ABB RAPID module: TCTM831_CYCLE_PATH_FOLLOW_CYCLE.mod

MODULE TCTM831_CYCLE_PATH_FOLLOW_CYCLE
    !*****************************************************
    !Project    : P21-100538 COJAFEX
    !Version:     1.0
    !Description:
    !Date:        04-2022
    !Author:      RLZ
    !*****************************************************
    !
    PERS pos OFFSET:=[0,0,0];
    PERS pos OFFSET_REF:=[0,0,0];
    PERS pos offsetprev:=[0,0,0];

    CONST num CALC_COUNTER:=71;             ! afstand tcp inductie ring - tcp lasers  55
    CONST num POS_FILTER_SIZE:=41;          ! oneven getal was 21
    CONST num ORIENT_FILTER_SIZE:=35;       ! oneven getal was 31
    CONST num PreStartLength:=90;           ! minimaal 2 * POS_FILTER_SIZE
    CONST num MaxLaserOutRange := 10;       ! als laser
    CONST num LaserDistMean := 15;          ! 15 laser datapunten worden gemiddeld voor het bepalen van einde buis (verkleining)
    CONST num EndTubeMinDistance := 12;     ! 20mm gemiddelde afstand verschil tussen de punten voor en de punten na is einde buis

    !PERS num nMovementCounter:=725;         ! Actual tcp heating ring position
    PERS num nPosFilterCounter:=704;        ! Calculated filtered pos position
    PERS num nOrientFilterCounter:=687;     ! Calculated filtered orient position
    PERS pos OrientVectorStart:=[-16.0742,645.886,223.213];
    PERS pos OrientVectorEind:=[-15.8133,665.273,253.56];
    PERS num Lasers{4}:=[-3449.93,-3441.27,-3504.93,-3514.26];
    PERS num nLaserData{4}:=[378.5,383,386.8,377];
    PERS num nLaserDataprev{4}:=[378.5,383,386.8,377];
    PERS num nLaserOutRange{4}:=[0,0,0,0];
    PERS bool END_TUBE_REACHED{2} := [FALSE, FALSE];

    PERS robtarget Assist1;
    PERS robtarget Assist2;
    PERS robtarget Assist3;
    PERS jointtarget joints;
    PERS num As1;
    PERS num As2;
    PERS num As3;
    PERS num As4;
    PERS num As5;
    PERS num As6;
    PERS num As7;

    PERS orient SaveLaserValue{10000};      ! Size should be the same as TargetNew
    PERS orient LaserDataAll{1200}:=[[0,0,0,0],
                                    [0,0,0,0],
                                    [0,0,0,0],
                                    [0,0,0,0],
                                    [0,0,0,0],
                                    [0,0,0,0],
                                    [0,0,0,0],
                                    [0,0,0,0],
                                    [0,0,0,0],
                                    [0,0,0,0],
                                    [0,0,0,0],
                                    [0,0,0,0],
                                    [0,0,0,0],
                                    [0,0,0,0],
                                    [0,0,0,0],
                                    [0,0,0,0],
                                    [0,0,0,0],
                                    [383.5,380.8,383.8,382.3],
                                    [383.5,380.9,383.9,382.2],
                                    [383.6,380.9,383.9,382.2],
                                    [383.6,381,383.8,382.1],
                                    [382.1,380.6,383.9,379.9],
                                    [382.1,380.6,383.9,379.9],
                                    [382.1,380.6,383.9,379.9],
                                    [382.1,380.6,383.8,379.9],
                                    [382.1,380.6,383.8,379.9],
                                    [382.1,380.5,383.7,380],
                                    [382.3,380.5,383.6,380.2],
                                    [382.3,380.3,383.8,380.2],
                                    [382.4,380.3,383.7,380.3],
                                    [382.4,380.4,383.5,380.2],
                                    [382.6,380.5,383.3,380.3],
                                    [382.6,380.6,383.5,380],
                                    [382.7,380.7,383.6,380.1],
                                    [382.8,380.6,383.5,380.1],
                                    [382.8,380.5,383.4,380],
                                    [382.9,380.6,383.3,380.1],
                                    [382.9,380.5,383.3,380.2],
                                    [383,380.4,383.3,380.3],
                                    [383,380.3,383.3,380.3],
                                    [383.1,380.5,383.1,380.3],
                                    [383.1,380.4,383.1,380.3],
                                    [383.2,380.2,383.1,380.4],
                                    [383.2,380.3,382.9,380.4],
                                    [383.2,380.2,383,380.3],
                                    [383.3,380.3,382.9,380.4],
                                    [383.4,380.3,383.1,380.2],
                                    [383.6,380.3,383.1,380.3],
                                    [383.4,380.2,383,380.3],
                                    [383.1,380.3,383.5,380.3],
                                    [383.2,380.3,383.4,380.3],
                                    [383.6,380.4,382.9,380.3],
                                    [383.9,380.3,382.5,380.4],
                                    [383.9,380.3,382.4,380.4],
                                    [383.9,380.4,382.5,380.4],
                                    [384,380.4,382.6,380.5],
                                    [384,380.3,382.6,380.5],
                                    [383,380.9,382.8,379.7],
                                    [383.1,381,382.5,379.4],
                                    [383.1,381.1,382.7,379.5],
                                    [383,381.2,382.7,379.4],
                                    [383,380.9,382.6,379.5],
                                    [382.6,380.7,382.8,379.7],
                                    [382.8,380.6,382.8,379.8],
                                    [382.9,380.3,382.5,380.2],
                                    [383,380.4,382.5,380.1],
                                    [383,380.5,382.8,380],
                                    [383.1,380.6,382.3,379.9],
                                    [383.1,380.6,382.3,379.9],
                                    [383.1,380.7,382.4,379.8],
                                    [383.2,380.6,382.6,379.9],
                                    [383.3,380.5,382.5,379.9],
                                    [383.3,380.5,382.4,380.1],
                                    [383.2,380.4,382.4,380.1],
                                    [383.4,380.3,382.3,380.2],
                                    [383.4,380.2,382.5,380.3],
                                    [383.3,380,382.4,380.3],
                                    [383.3,380.1,382.4,380.4],
                                    [383.6,380,382.6,380.3],
                                    [383.6,380,382.3,380.3],
                                    [383.4,380,382.4,380.4],
                                    [383.4,380.1,382.3,380.5],
                                    [383.3,380,382.3,380.2],
                                    [383.3,380.2,382.3,380.3],
                                    [383.3,380.2,382.5,380.2],
                                    [383.3,380.2,382.6,380.3],
                                    [383.2,380.1,382.4,380.3],
                                    [383.1,380.2,382.5,380.2],
                                    [383,380.1,382.7,380.2],
                                    [383,380.2,382.4,380.1],
                                    [383.1,380.4,383,380],
                                    [382.8,380.3,383.1,380.1],
                                    [382.5,380.4,383.1,379.9],
                                    [382.5,380.5,383.6,379.6],
                                    [382.4,380.7,383.4,379.6],
                                    [382.3,380.9,383.8,379.3],
                                    [382.2,381,383.5,379.2],
                                    [382,381,383.7,379.2],
                                    [381.8,381.1,383.8,379.1],
                                    [381.6,381.3,384.2,378.9],
                                    [381.3,381.3,384.4,378.9],
                                    [381.2,381.4,384.6,378.8],
                                    [381.1,381.4,384.5,378.6],
                                    [380.9,381.6,384.6,378.5],
                                    [380.8,381.6,384.8,378.4],
                                    [380.6,381.7,385.1,378.5],
                                    [380.2,381.9,385.4,378.3],
                                    [380,382.2,385.6,378.2],
                                    [379.7,382.1,385.8,378.2],
                                    [379.4,382.1,386.1,378.2],
                                    [379.5,381.7,386.3,378.2],
                                    [379.5,381.9,386.1,378.4],
                                    [379.5,381.7,386.1,378.4],
                                    [379.5,381.5,386.2,378.6],
                                    [379.3,381.5,386.2,378.6],
                                    [379.3,381.5,386.4,378.6],
                                    [379.3,381.4,386.4,378.6],
                                    [379.2,381.2,386.6,378.7],
                                    [379.1,381.5,386.4,378.9],
                                    [379.1,381.3,386.6,378.8],
                                    [379.1,381.2,386.6,378.9],
                                    [379,381.5,386.5,378.9],
                                    [379,381.4,386.4,378.7],
                                    [378.9,381.3,386.4,378.8],
                                    [378.9,381.2,386.2,379.1],
                                    [378.8,381.1,386.5,378.9],
                                    [378.7,381.1,386.6,378.9],
                                    [378.6,381.2,386.7,379],
                                    [378.5,381.4,386.7,378.8],
                                    [378.5,381.3,386.7,378.8],
                                    [378.4,381.3,387.4,378.8],
                                    [378.4,381.4,387.3,378.6],
                                    [378.3,381.5,387.1,378.6],
                                    [378.3,381.4,387.1,378.5],
                                    [378.2,381.5,387.2,378.5],
                                    [378.4,381.7,387.1,378.4],
                                    [378.4,381.7,387.2,378.4],
                                    [378.3,381.9,387.2,378.3],
                                    [378.2,381.8,387.3,378.2],
                                    [378.3,381.8,387.3,378.1],
                                    [378.1,381.9,387.1,378.2],
                                    [378.3,381.8,387.2,378.2],
                                    [378.2,382,387.3,378.2],
                                    [378.2,382.1,387.3,378.1],
                                    [378.2,382,387.1,378.1],
                                    [378.2,382.1,387,377.9],
                                    [378.2,382.1,387.1,378],
                                    [378.2,382.1,387.4,378],
                                    [378.2,382,387,378.1],
                                    [378.2,382.1,387.6,378],
                                    [378.2,382.1,387.2,378.1],
                                    [378.3,382.2,387.1,378],
                                    [378.3,382.1,387.1,377.9],
                                    [378.3,382.3,387.4,378],
                                    [378.3,382.1,387.1,378],
                                    [378.4,382,387.1,378],
                                    [378.4,381.9,386.9,378.1],
                                    [378.4,382.1,387,378],
                                    [378.4,382,387.2,378.2],
                                    [378.3,382.2,387.1,378.2],
                                    [378.4,382.2,387,378.1],
                                    [378.5,382.1,386.9,378.1],
                                    [378.5,382,387.1,378.2],
                                    [378.5,382,387,378.2],
                                    [378.5,382,386.9,378.1],
                                    [378.6,382,386.7,378.1],
                                    [378.6,382,386.8,378],
                                    [378.6,382,386.9,378.1],
                                    [378.6,382,387.1,378.1],
                                    [378.5,382.1,387.1,378],
                                    [378.5,382.2,386.9,377.9],
                                    [378.5,382.2,386.9,377.9],
                                    [378.6,382.2,387.1,377.9],
                                    [378.6,382.3,387.1,377.8],
                                    [378.6,382.5,387,377.9],
                                    [378.6,382.2,386.7,377.9],
                                    [378.5,382.1,386.8,377.8],
                                    [378.5,382.2,386.9,377.9],
                                    [378.5,382.3,387,377.9],
                                    [378.5,382.3,387.3,377.8],
                                    [378.5,382.2,387.2,377.8],
                                    [378.4,382.3,387.2,377.8],
                                    [378.4,382.3,387.3,377.7],
                                    [378.3,382.3,387.4,377.7],
                                    [378.2,382.4,387.4,377.7],
                                    [378.2,382.3,387.5,377.8],
                                    [378,382.3,387.4,377.8],
                                    [378.1,382.3,387.3,377.8],
                                    [378.1,382.3,387.5,377.8],
                                    [378,382.3,387.6,377.8],
                                    [378,382.4,387.7,377.8],
                                    [378,382.4,387.6,377.9],
                                    [377.9,382.3,387.6,377.8],
                                    [377.9,382.4,387.6,377.8],
                                    [377.9,382.2,387.4,377.8],
                                    [377.8,382.2,387.8,377.8],
                                    [377.8,382.2,387.8,377.9],
                                    [377.7,382.2,387.8,377.9],
                                    [377.8,382.1,387.8,378],
                                    [377.7,382.1,387.8,378],
                                    [377.8,382.1,387.8,378],
                                    [377.7,382,387.6,378.2],
                                    [377.6,382,387.8,378.3],
                                    [377.7,381.9,387.7,378.3],
                                    [377.7,381.6,387.7,378.5],
                                    [377.6,381.7,388,378.4],
                                    [377.7,381.8,388,378.5],
                                    [377.6,381.9,387.9,378.4],
                                    [377.5,381.7,387.7,378.4],
                                    [377.5,381.7,387.9,378.5],
                                    [377.5,381.6,387.9,378.6],
                                    [377.5,381.6,388.1,378.6],
                                    [377.4,381.5,387.9,378.7],
                                    [377.4,381.5,387.9,378.7],
                                    [377.3,381.4,388.2,378.7],
                                    [377.3,381,388.2,378.9],
                                    [377.1,381.5,388.3,378.7],
                                    [377.1,381.6,388.4,378.7],
                                    [377,381.6,388.5,378.7],
                                    [377,381.7,388.6,378.8],
                                    [377,381.4,388.3,378.8],
                                    [376.9,381.5,388.7,378.7],
                                    [376.9,381.4,388.7,378.8],
                                    [376.8,381.5,388.6,378.8],
                                    [376.9,381.5,388.6,378.8],
                                    [376.8,381.7,388.6,378.6],
                                    [376.9,381.6,388.6,378.8],
                                    [376.9,381.5,388.7,378.8],
                                    [376.8,381.5,388.7,378.7],
                                    [376.8,381.5,388.9,378.8],
                                    [376.8,381.7,389,378.7],
                                    [376.6,381.8,389,378.7],
                                    [376.7,381.7,388.8,378.7],
                                    [376.7,381.7,388.8,378.6],
                                    [376.7,381.7,389.1,378.7],
                                    [376.5,381.5,388.9,378.7],
                                    [375.7,381.8,389.8,378.6],
                                    [375.2,382,390.2,378.5],
                                    [375.7,381.9,390.1,378.5],
                                    [375.3,382.1,390.2,378.4],
                                    [375.5,381.8,390.1,378.6],
                                    [375.4,382,390.4,378.5],
                                    [375.3,382,390.2,378.6],
                                    [375.2,381.8,390.4,378.6],
                                    [375.3,381.9,390.3,378.5],
                                    [375.3,382.1,390,378.3],
                                    [375.3,381.9,390,378.4],
                                    [375.2,382.1,390.4,378.4],
                                    [375.3,381.9,389.9,378.5],
                                    [375.3,381.9,389.9,378.5],
                                    [375.2,382,390,378.6],
                                    [375.2,381.8,390.4,378.6],
                                    [375.1,381.9,390.4,378.5],
                                    [375.2,381.9,390.3,378.6],
                                    [375,381.8,390.6,378.6],
                                    [375.1,381.9,390.4,378.7],
                                    [375,381.8,390.5,378.7],
                                    [375.1,381.7,390.5,378.8],
                                    [375,381.9,390.7,378.7],
                                    [375.1,381.8,390.5,378.6],
                                    [375,381.8,390.5,378.7],
                                    [375,381.9,390.3,378.7],
                                    [375,381.8,390.5,378.7],
                                    [375.2,381.7,390.7,378.7],
                                    [376.3,381.5,389.3,378.9],
                                    [375.9,381.6,389.7,378.8],
                                    [375.6,381.6,389.8,378.9],
                                    [375.6,381.6,390,378.8],
                                    [375.2,381.6,390.3,378.9],
                                    [374.9,381.5,390.6,378.9],
                                    [374.8,381.4,390.9,378.9],
                                    [374.5,381.7,391,378.8],
                                    [374.3,381.8,391.1,378.8],
                                    [374.5,381.8,390.9,378.8],
                                    [374.6,381.6,391.1,378.9],
                                    [374.7,381.8,390.8,378.8],
                                    [375,381.6,390.8,378.8],
                                    [376.4,381.3,389.3,379],
                                    [376.5,381.4,389.1,378.9],
                                    [376,381.4,389.7,378.9],
                                    [375.9,381.5,389.5,379],
                                    [375.6,381.5,390,378.8],
                                    [376.7,381.3,389.1,378.9],
                                    [376,381.6,389.6,378.7],
                                    [376.4,381.4,389.3,378.8],
                                    [375.9,381.5,390,378.8],
                                    [375.7,381.4,390.2,378.8],
                                    [376.9,381.1,388.7,379.1],
                                    [376.5,381.4,389.3,378.8],
                                    [376.7,381.5,389.2,378.8],
                                    [376.4,381.3,389.5,378.9],
                                    [376.3,381.4,389.5,379],
                                    [376.5,381.2,389.4,379],
                                    [376.5,381.1,389.3,379.2],
                                    [377.5,380.9,388.1,379.3],
                                    [377,381.3,388.9,378.9],
                                    [377.1,381.4,388.8,378.9],
                                    [376.8,381.2,389.2,379.1],
                                    [376.5,381.3,389.4,378.9],
                                    [377.5,381,388.4,379.2],
                                    [377.2,381.2,388.6,379],
                                    [377.5,381.1,388.3,379],
                                    [377.1,381.1,388.9,379.2],
                                    [376.9,381.2,389,379],
                                    [377,381.1,388.9,379.1],
                                    [376.8,381.2,389.1,379.1],
                                    [377.1,381.2,388.6,379.1],
                                    [377,381,388.8,379.1],
                                    [377.8,380.9,388.1,379.2],
                                    [378.2,380.9,387.7,379.3],
                                    [377.6,381,388.4,379.1],
                                    [377.3,381.5,388.6,378.8],
                                    [377.7,381.1,388.3,379.1],
                                    [377.1,381.5,389,378.7],
                                    [377.2,381.5,388.8,378.9],
                                    [377.1,381.5,388.9,378.9],
                                    [376.9,381.5,388.9,378.8],
                                    [377,381.4,389,379],
                                    [377.1,381.4,388.9,378.9],
                                    [377,381.4,388.9,379],
                                    [377.2,381.2,388.7,379],
                                    [377.1,381.4,388.7,378.8],
                                    [377.2,381.2,388.8,379],
                                    [377.1,381.4,388.9,378.9],
                                    [377.2,381.2,388.9,379],
                                    [377.1,381.3,388.8,379],
                                    [377.1,381.1,388.7,379],
                                    [377,381.1,388.7,379.1],
                                    [377.2,381.3,388.5,379],
                                    [377.1,381.4,388.7,378.9],
                                    [377.3,381.3,388.4,379.1],
                                    [377.2,381.6,388.5,378.9],
                                    [377.3,381.3,388.4,379.2],
                                    [377.1,381.5,388.6,378.9],
                                    [377.5,381.2,388.3,379.1],
                                    [377.2,381.3,388.6,379],
                                    [377.4,381.1,388.4,379.3],
                                    [377.3,381.2,388.3,379.2],
                                    [377.1,381,388.4,379.2],
                                    [377.2,381,388.6,379.3],
                                    [377,381.2,388.6,379.2],
                                    [377,381,388.5,379.4],
                                    [376.9,381,388.7,379.3],
                                    [376.9,381.1,388.7,379.4],
                                    [376.9,381,388.8,379.3],
                                    [376.8,381.1,388.9,379.3],
                                    [376.9,381.1,388.7,379.4],
                                    [376.7,381.2,388.9,379.2],
                                    [376.9,381,388.5,379.4],
                                    [376.7,381.2,389,379.3],
                                    [376.7,381,388.8,379.4],
                                    [376.6,381.1,389,379.3],
                                    [376.4,381.2,389.2,379.3],
                                    [376.3,381.1,389.6,379.4],
                                    [376.3,381.1,389.4,379.4],
                                    [376.3,381.2,389.5,379.5],
                                    [376.3,381.2,389,379.4],
                                    [376.5,381,389.1,379.5],
                                    [376.4,381.2,389.3,379.4],
                                    [376.6,381.1,389.2,379.4],
                                    [376.5,381.2,389.2,379.4],
                                    [376.6,381.1,389.1,379.4],
                                    [376.4,381.1,389.2,379.5],
                                    [377.3,380.6,388.2,379.8],
                                    [377.2,381.1,388.5,379.3],
                                    [377.3,381.1,388.4,379.4],
                                    [376.5,381.3,388.9,379.2],
                                    [376.6,381.4,389,379.1],
                                    [376.4,381.1,389,379.4],
                                    [376.1,381.3,389.5,379.2],
                                    [377.3,380.8,388.4,379.7],
                                    [376.8,381.3,388.9,379.2],
                                    [377.2,381,388.4,379.4],
                                    [376.6,381.4,388.9,379.2],
                                    [376.7,381.3,388.8,379.1],
                                    [376.6,381.3,389.1,379.2],
                                    [376.6,381.1,389.2,379.4],
                                    [376.6,381.2,389,379.4],
                                    [376.4,381.1,389.2,379.4],
                                    [376.4,381.1,389.1,379.4],
                                    [376.5,381.3,389,379.3],
                                    [376.4,381.2,389,379.3],
                                    [376.5,381.2,389.1,379.4],
                                    [376.5,381.1,389.2,379.5],
                                    [376.6,380.9,389.1,379.5],
                                    [376.5,381,389.1,379.4],
                                    [376.6,380.8,389.1,379.7],
                                    [377.8,380.7,387.8,379.9],
                                    [376.9,381,388.8,379.2],
                                    [376.9,381,388.6,379.4],
                                    [376.7,381.1,388.8,379.5],
                                    [376.7,381.1,388.7,379.5],
                                    [376.8,381.2,388.7,379.3],
                                    [376.7,381,388.7,379.5],
                                    [376.5,381.4,388.8,379.1],
                                    [376.6,381.3,388.8,379.3],
                                    [376.2,381.4,389.2,379.1],
                                    [376.1,381.5,389.1,379.1],
                                    [376,381.3,389.3,379.3],
                                    [376,381.3,389.5,379.2],
                                    [376,381.2,389.4,379.4],
                                    [375.9,381.3,389.6,379.2],
                                    [376.2,381.2,389,379.4],
                                    [376,381.3,389.7,379.2],
                                    [376.3,381.1,389.4,379.4],
                                    [376.1,381.1,389.4,379.3],
                                    [376.9,380.8,388.6,379.6],
                                    [376.9,381.2,388.4,379.3],
                                    [377.2,381.1,388.4,379.4],
                                    [376.5,381.3,388.9,379.3],
                                    [376.7,381.3,388.7,379.2],
                                    [376.5,381,389.1,379.5],
                                    [376.3,381.2,389.2,379.3],
                                    [376.3,381.1,389.1,379.4],
                                    [376.4,381.1,389.2,379.3],
                                    [376.5,381.1,389.2,379.4],
                                    [376.3,381.1,389,379.5],
                                    [377.4,380.8,388.2,379.7],
                                    [377.4,380.9,388.2,379.5],
                                    [377.3,381,388.4,379.4],
                                    [376.9,381.2,388.8,379.3],
                                    [377,381.2,388.4,379.2],
                                    [376.9,381.1,388.6,379.4],
                                    [377,381.1,388.6,379.5],
                                    [376.6,381.2,388.7,379.3],
                                    [376.8,381.1,388.6,379.5],
                                    [376.6,381.1,388.7,379.4],
                                    [376.5,381.2,389.1,379.4],
                                    [376.6,381.2,389.2,379.6],
                                    [376.5,381.1,389.3,379.5],
                                    [376.6,381.2,388.9,379.4],
                                    [376.6,381.1,389,379.4],
                                    [377.4,380.8,388.1,379.7],
                                    [377.3,381.1,388.2,379.3],
                                    [377.4,380.9,388.3,379.5],
                                    [376.8,381.3,388.7,379.2],
                                    [376.8,381.4,389,379.1],
                                    [376.7,381.4,389.1,379.2],
                                    [376.5,381.4,388.9,379.2],
                                    [376.6,381.3,389.2,379.3],
                                    [377.4,380.7,388.2,379.9],
                                    [377.7,381,388,379.4],
                                    [377.2,381.3,388.4,379.4],
                                    [377.3,381.5,388.6,379.1],
                                    [376.9,381.5,388.7,379.1],
                                    [376.7,381.5,388.8,378.9],
                                    [376.7,381.4,388.8,379.1],
                                    [376.5,381.3,389.2,379.2],
                                    [376.5,381.4,389,379.1],
                                    [376.3,381.4,389.3,379.1],
                                    [376.2,381.3,389.1,379.3],
                                    [376.4,381.2,389.1,379.2],
                                    [377.4,381.1,388.1,379.4],
                                    [377.9,381.2,387.6,379.2],
                                    [378.2,381.1,387.2,379.3],
                                    [378.7,381,386.9,379.4],
                                    [378.5,381.1,387,379.3],
                                    [378.6,381.1,386.9,379.3],
                                    [378.5,381.1,387.4,379.3],
                                    [378.4,381.1,387.4,379.2],
                                    [378.5,381.1,387.1,379.3],
                                    [378.4,381.1,387,379.3],
                                    [378.4,381.2,387.1,379.2],
                                    [378.6,381.1,387.1,379.2],
                                    [378.5,381.1,387.4,379.2],
                                    [378.4,381.2,387.2,379.2],
                                    [377.1,381.4,388.6,378.9],
                                    [377.6,381.3,388.1,379],
                                    [377.8,381.4,388.1,378.9],
                                    [378.3,381.4,387.5,379],
                                    [378.7,381.3,386.9,379],
                                    [379,381.3,386.6,379.1],
                                    [379.1,381.3,386.7,379.1],
                                    [378.9,381.3,386.8,379],
                                    [378.8,381.3,387,379],
                                    [378.7,381.5,387.1,378.9],
                                    [378.5,381.6,387.1,378.8],
                                    [378.5,381.5,387.1,378.8],
                                    [378.4,381.4,387.6,378.8],
                                    [377.1,381.8,388.8,378.6],
                                    [376.6,381.7,389.3,378.7],
                                    [377.1,381.7,388.7,378.6],
                                    [377.1,381.7,388.6,378.7],
                                    [377.2,381.7,388.3,378.7],
                                    [377.3,381.7,388.4,378.8],
                                    [377.4,382.1,388.2,378.8],
                                    [377.5,381.8,387.9,378.6],
                                    [378.2,381.6,387.2,378.8],
                                    [377.7,381.7,387.9,378.6],
                                    [377.7,381.5,387.9,378.9],
                                    [377.4,381.6,388.3,378.7],
                                    [377.5,381.6,388.1,378.9],
                                    [377.2,381.4,388.3,378.9],
                                    [377.2,381.6,388.6,378.7],
                                    [377.4,381.8,388.5,378.7],
                                    [377.2,381.5,388.5,379],
                                    [376.9,381.8,388.7,378.7],
                                    [377.2,381.8,388.5,378.8],
                                    [376.6,381.8,389.2,378.7],
                                    [377,381.5,388.6,378.8],
                                    [378.6,380.7,387.2,379.7],
                                    [377.9,381,387.5,379.3],
                                    [378,381.1,387.5,379.2],
                                    [377.8,381.1,387.7,379.1],
                                    [377.8,381.3,387.6,379],
                                    [377.7,381.5,387.7,378.8],
                                    [377.7,381.7,388,378.7],
                                    [377.8,382,388,378.4],
                                    [377.7,382,387.9,378.4],
                                    [377.7,382,387.9,378.4],
                                    [377.6,382,387.9,378.5],
                                    [377.6,381.7,388,378.6],
                                    [377.6,381.8,387.9,378.5],
                                    [377.6,381.7,388,378.8],
                                    [377.6,381.6,387.8,378.8],
                                    [377.6,381.5,388.1,378.7],
                                    [377.5,381.5,387.9,378.7],
                                    [376.9,381.7,388.6,378.7],
                                    [377.5,381.5,388,378.9],
                                    [377.5,381.6,387.9,378.8],
                                    [377.4,381.7,387.9,378.7],
                                    [377.4,381.6,388.1,378.8],
                                    [377.4,381.5,388.1,378.8],
                                    [377.4,381.6,387.8,378.7],
                                    [377.5,381.5,387.9,378.8],
                                    [377.5,381.6,387.9,378.7],
                                    [377.6,381.7,387.8,378.8],
                                    [377.6,381.7,387.9,378.7],
                                    [377.6,381.6,387.8,378.7],
                                    [377.5,381.8,388,378.7],
                                    [376.8,381.9,388.7,378.6],
                                    [376.1,382.2,389.5,378.4],
                                    [376.7,381.9,388.8,378.6],
                                    [376.5,382,388.9,378.5],
                                    [376.9,381.9,388.5,378.6],
                                    [376.9,382,388.9,378.5],
                                    [377,381.9,388.7,378.6],
                                    [377.1,381.8,388.4,378.6],
                                    [377.2,381.7,388.4,378.6],
                                    [377.2,381.8,388.2,378.7],
                                    [377.2,381.8,388.3,378.6],
                                    [377.3,381.8,388.2,378.5],
                                    [377.3,381.7,388.5,378.6],
                                    [377.4,381.9,388.6,378.4],
                                    [377.4,381.8,388.3,378.6],
                                    [378.7,381.4,386.9,378.9],
                                    [378.9,381.3,386.5,378.9],
                                    [378.5,381.4,387.1,378.7],
                                    [378.2,381.7,387.2,378.6],
                                    [378,381.8,387.8,378.5],
                                    [377.9,381.8,387.8,378.4],
                                    [377.8,381.9,387.8,378.5],
                                    [377.6,381.9,387.9,378.4],
                                    [377.5,381.8,388.2,378.6],
                                    [377.5,381.6,388.2,378.6],
                                    [377.5,381.6,388.1,378.7],
                                    [377.4,381.6,387.9,378.8],
                                    [377.3,381.4,388.2,378.8],
                                    [377.3,381.5,388.6,378.6],
                                    [377.5,381.5,388.2,378.5],
                                    [377.5,381.8,388,378.4],
                                    [377.5,382,388.1,378.3],
                                    [377.5,382.1,388.2,378.2],
                                    [377.7,382.1,388,378.2],
                                    [377.7,382,387.8,378.2],
                                    [377.7,381.9,387.8,378.2],
                                    [377.8,382.1,388,378.1],
                                    [377.8,382.1,387.9,378.2],
                                    [377.8,382.2,387.7,378.1],
                                    [377.8,382.1,387.7,378.2],
                                    [377.8,381.8,387.6,378.1],
                                    [377.9,382,387.7,378.2],
                                    [378,382.1,387.6,378],
                                    [378.1,382.3,387.5,378],
                                    [378.2,382.4,387.4,377.8],
                                    [378.4,382.6,387.2,377.5],
                                    [378.4,382.7,387.3,377.3],
                                    [378.4,382.4,387.1,377.6],
                                    [378.4,382.4,387.1,377.8],
                                    [378.3,382.2,387,377.9],
                                    [378.3,382.3,387,377.9],
                                    [378.4,382.2,387,378],
                                    [378.4,382.2,387,378],
                                    [378.6,382,387.1,378.2],
                                    [378.6,381.9,386.8,378.2],
                                    [378.6,382.2,387,378.1],
                                    [378.6,382.1,386.8,378.1],
                                    [378.6,382.2,387,378],
                                    [378.6,382.3,386.8,378.1],
                                    [378.7,381.9,386.8,378],
                                    [378.8,382,386.8,378.1],
                                    [378.9,382,386.8,378.1],
                                    [378.9,382,386.7,378],
                                    [379.1,382,386.8,378.1],
                                    [379.1,382,386.6,378.1],
                                    [378.9,382,386.4,378],
                                    [379,382,386.4,378],
                                    [379,382,386.5,378],
                                    [379.1,382.1,386.5,377.9],
                                    [379,382,386.4,377.9],
                                    [379.1,382.1,386.4,377.8],
                                    [379.1,382.2,386.5,377.9],
                                    [379,382.2,386.3,377.9],
                                    [379.1,382.3,386.4,377.7],
                                    [379.1,382.2,386.3,377.8],
                                    [379,382.2,386.4,377.9],
                                    [379,382.2,386.4,377.8],
                                    [378.9,382.2,386.8,377.7],
                                    [379,382.3,386.3,377.6],
                                    [378.9,382.5,386.6,377.5],
                                    [378.9,382.6,386.5,377.5],
                                    [378.8,382.6,386.7,377.4],
                                    [378.8,382.7,386.6,377.5],
                                    [378.8,382.8,386.6,377.3],
                                    [378.8,382.7,386.7,377.4],
                                    [378.8,382.7,386.8,377.3],
                                    [378.8,382.8,386.6,377.4],
                                    [378.5,382.7,386.8,377.2],
                                    [378.4,382.5,387.1,377.4],
                                    [378.3,382.4,386.9,377.5],
                                    [378.1,382.1,387.2,377.6],
                                    [378,382.3,387.4,377.7],
                                    [378.2,382.5,387.3,377.5],
                                    [378.2,382.5,387.3,377.4],
                                    [378.1,382.7,387.2,377.2],
                                    [378.2,382.9,387.1,377.1],
                                    [378.2,382.9,387.2,377],
                                    [378.3,383.1,387.1,376.7],
                                    [378.5,383.3,387,376.6],
                                    [378.5,383.5,386.7,376.5],
                                    [378.4,383.5,386.9,376.6],
                                    [378.2,383.2,387.2,376.8],
                                    [378.2,383.1,387.1,376.8],
                                    [378.1,383.1,387.2,376.9],
                                    [378.2,383,387.1,377],
                                    [378.1,382.9,387.5,377],
                                    [378,383,387.4,377],
                                    [377.9,383.1,387.2,377],
                                    [378,383,387.3,377.1],
                                    [378.1,382.9,387.4,377.1],
                                    [377.9,382.8,387.3,377.1],
                                    [377.9,383,387.2,377.1],
                                    [377.9,382.9,387.1,377.2],
                                    [377.8,383,387.2,377.1],
                                    [377.9,382.8,387.3,377.1],
                                    [377.9,382.9,387.3,377.1],
                                    [377.9,382.9,387.3,377.1],
                                    [377.8,382.9,387.3,377.3],
                                    [377.8,382.7,387.2,377.4],
                                    [377.7,382.5,387.5,377.6],
                                    [377.5,382.5,387.6,377.7],
                                    [377.5,382.4,387.3,377.7],
                                    [377.7,382.5,387.5,377.7],
                                    [377.7,382.6,387.4,377.5],
                                    [377.9,382.7,387.5,377.4],
                                    [377.9,382.7,387.1,377.3],
                                    [378,382.8,387.2,377.3],
                                    [378.1,382.8,386.9,377.2],
                                    [378.1,382.9,387.1,377.2],
                                    [378.2,382.9,387.2,377.2],
                                    [378.1,382.9,387,377.2],
                                    [378.2,382.9,386.9,377.1],
                                    [378.2,383,386.8,377.2],
                                    [378.3,383,387,377.1],
                                    [378.3,383,386.8,377.1],
                                    [378.3,383.2,387,376.9],
                                    [378.4,383.2,386.8,376.8],
                                    [378.5,383.3,386.8,376.7],
                                    [378.6,383.3,386.7,376.7],
                                    [378.5,383.3,386.6,376.7],
                                    [378.5,383.1,386.9,376.9],
                                    [378.4,383,387.1,377.1],
                                    [378.3,382.9,387.1,377.1],
                                    [378.5,383,386.8,377],
                                    [379,383.3,386.4,376.6],
                                    [379,383.4,386.2,376.6],
                                    [379,383.4,386.3,376.7],
                                    [379,383.4,386.3,376.7],
                                    [379,383.4,386.4,376.6],
                                    [379,383.4,386.3,376.7],
                                    [378.9,383.4,386.2,376.6],
                                    [378.9,383.4,386.2,376.6],
                                    [378.9,383.4,386.2,376.7],
                                    [379.1,383.4,386.2,376.7],
                                    [379,383.4,386.1,376.6],
                                    [379,383.4,386.3,376.5],
                                    [379.1,383.3,386,376.6],
                                    [379.1,383.4,386.2,376.5],
                                    [379.1,383.5,386.5,376.5],
                                    [379.1,383.4,386.2,376.5],
                                    [379.1,383.3,386.3,376.6],
                                    [379.1,383.4,386.3,376.5],
                                    [379.1,383.4,386.2,376.5],
                                    [379.1,383.4,386.1,376.6],
                                    [379.2,383.4,386.3,376.6],
                                    [379.3,383.4,386.2,376.5],
                                    [379.2,383.4,386.2,376.4],
                                    [379.1,383.5,386.1,376.4],
                                    [379.2,383.5,386.1,376.5],
                                    [379.2,383.6,386,376.4],
                                    [379.2,383.6,385.9,376.3],
                                    [379.3,383.6,385.9,376.3],
                                    [379.2,383.5,386,376.4],
                                    [379.2,383.6,386.1,376.3],
                                    [379.2,383.5,385.9,376.3],
                                    [379.2,383.7,385.8,376.3],
                                    [379.2,383.7,385.9,376.4],
                                    [379.3,383.7,386,376.3],
                                    [379.3,383.6,385.9,376.2],
                                    [379.3,383.7,386.1,376.3],
                                    [379.3,383.6,385.9,376.4],
                                    [379.3,383.7,385.9,376.3],
                                    [379.2,383.6,386.1,376.3],
                                    [379.2,383.6,386.1,376.3],
                                    [379.1,383.7,386,376.3],
                                    [379.3,383.6,385.9,376.3],
                                    [379.2,383.5,385.6,376.4],
                                    [379.2,383.6,385.9,376.3],
                                    [379.3,383.5,385.8,376.4],
                                    [379.2,383.5,385.8,376.4],
                                    [379.2,383.5,385.9,376.4],
                                    [379.1,383.6,386,376.4],
                                    [379.3,383.4,385.9,376.6],
                                    [379.1,383.4,385.9,376.5],
                                    [379.1,383.4,385.9,376.6],
                                    [379.1,383.4,386.1,376.5],
                                    [379,383.3,386,376.5],
                                    [379,383.3,386,376.6],
                                    [379,383.3,386.1,376.6],
                                    [379.1,383.4,385.9,376.6],
                                    [379,383.4,386.2,376.6],
                                    [379,383.4,385.8,376.7],
                                    [379.1,383.3,385.8,376.6],
                                    [379.1,383.4,385.8,376.6],
                                    [379.2,383.4,385.9,376.6],
                                    [379.2,383.3,385.9,376.7],
                                    [379.1,383.4,385.9,376.7],
                                    [379.2,383.4,385.9,376.6],
                                    [379.2,383.4,385.7,376.7],
                                    [379.4,383.3,386,376.7],
                                    [379.4,383.3,385.8,376.7],
                                    [379.4,383.2,385.6,376.6],
                                    [379.5,383.2,385.4,376.7],
                                    [379.6,383.2,385.6,376.8],
                                    [379.7,383.4,385.6,376.7],
                                    [379.6,383.3,385.5,376.7],
                                    [379.7,383.4,385.5,376.7],
                                    [379.6,383.2,385.5,376.8],
                                    [379.8,383.3,385.6,376.8],
                                    [379.8,383.2,385.3,376.8],
                                    [380,383.2,385.1,376.9],
                                    [380.2,383.2,385.2,376.8],
                                    [380.1,383.1,385.2,376.9],
                                    [380.1,383,385.2,376.9],
                                    [380.1,383,385.1,377],
                                    [380.2,383,385.1,377.1],
                                    [380.2,382.9,385,377],
                                    [380,382.9,385,377.1],
                                    [380,382.8,385,377.1],
                                    [380.2,382.8,384.8,377.1],
                                    [380.3,382.7,384.9,377.1],
                                    [380.4,382.6,384.7,377.1],
                                    [380.3,382.7,384.6,377.1],
                                    [380.5,382.7,384.7,377.2],
                                    [380.5,382.6,384.6,377.1],
                                    [380.4,382.7,384.5,377.1],
                                    [380.4,382.5,384.3,377.2],
                                    [380.6,382.4,384.3,377.2],
                                    [380.5,382.4,384.2,377.3],
                                    [380.3,382.3,384.5,377.2],
                                    [380.6,382.2,384.4,377],
                                    [380.8,382.1,384,377.4],
                                    [380.7,382.1,384.1,377.3],
                                    [380.8,382.2,384.1,377.4],
                                    [380.8,382,384.2,377.4],
                                    [380.9,381.9,383.9,377.6],
                                    [380.9,381.9,384,377.5],
                                    [380.9,381.8,383.7,377.5],
                                    [380.9,381.7,383.6,377.7],
                                    [381,381.6,383.5,377.8],
                                    [380.7,381.8,384,377.7],
                                    [380.9,381.6,383.7,377.7],
                                    [380.9,381.5,383.9,377.8],
                                    [381,381.6,383.7,377.8],
                                    [381,381.5,383.9,377.8],
                                    [381.1,381.5,383.8,377.8],
                                    [381.1,381.5,383.6,377.9],
                                    [381.1,381.4,383.7,377.9],
                                    [381.2,381.5,383.6,377.9],
                                    [381.2,381.3,383.7,377.9],
                                    [381.2,381.3,383.6,378],
                                    [381.1,381.3,383.7,378],
                                    [381.1,381.3,383.8,378.1],
                                    [381.1,381.2,383.6,378],
                                    [381,381.3,383.7,378.1],
                                    [381,381.1,383.8,378.1],
                                    [381,381.2,383.7,378.1],
                                    [380.9,381.1,383.9,378.1],
                                    [380.8,381.1,383.6,378.1],
                                    [380.8,381.2,383.9,378.1],
                                    [380.8,381.1,383.9,378.1],
                                    [380.7,381,384,378.1],
                                    [380.7,380.9,384,378.1],
                                    [380.7,381,384.3,378.1],
                                    [380.8,381,383.7,378],
                                    [380.7,380.8,383.6,378],
                                    [380.9,380.9,383.9,378],
                                    [380.8,380.9,383.7,378.1],
                                    [380.8,380.7,383.8,378.1],
                                    [380.7,380.9,384,378.2],
                                    [380.7,380.9,383.8,378.1],
                                    [380.8,380.8,383.8,378.1],
                                    [380.8,381,383.7,377.9],
                                    [380.7,381.1,383.6,377.9],
                                    [380.7,381.1,383.7,377.8],
                                    [380.5,381.3,383.6,377.7],
                                    [380.7,381.4,383.8,377.4],
                                    [380.5,381.4,383.8,377.5],
                                    [380.7,381.1,383.9,377.7],
                                    [380.8,381.1,383.7,377.7],
                                    [380.9,381,384,377.8],
                                    [380.9,380.9,383.6,377.9],
                                    [380.8,380.9,383.5,378],
                                    [380.9,380.8,383.5,378],
                                    [381,380.8,383.5,378],
                                    [380.9,380.8,383.8,378.1],
                                    [380.9,380.8,383.6,378.1],
                                    [381,380.7,383.4,378.1],
                                    [381,380.7,383.6,378.1],
                                    [381.1,380.6,383.6,378.2],
                                    [381.1,380.7,383.6,378.1],
                                    [381.3,380.6,383.6,378.3],
                                    [381.1,380.6,383.4,378.2],
                                    [381.2,380.5,383.5,378.4],
                                    [381.2,380.4,383.5,378.4],
                                    [381.3,380.6,383.5,378.4],
                                    [381.3,380.4,383.3,378.4],
                                    [381.3,380.3,383.1,378.4],
                                    [381.3,380.3,383.1,378.6],
                                    [381.5,380.4,383.2,378.5],
                                    [381.5,380.2,383.3,378.6],
                                    [381.7,380.2,383,378.6],
                                    [381.7,380.2,383.2,378.7],
                                    [381.8,380.1,382.9,378.8],
                                    [381.9,380,382.9,378.9],
                                    [382,379.9,382.7,379],
                                    [382,379.9,382.8,379],
                                    [381.9,380,382.9,379],
                                    [382.1,379.9,382.8,379],
                                    [382,379.8,382.7,379.2],
                                    [382.2,379.6,383,379.3],
                                    [382.3,379.6,382.5,379.3],
                                    [382.3,379.6,382.4,379.4],
                                    [382.4,379.7,382.6,379.3],
                                    [382.4,379.5,382,379.5],
                                    [382.5,379.3,382.4,379.6],
                                    [382.6,379.3,382.5,379.7],
                                    [382.6,379.3,382.4,379.6],
                                    [382.6,379.2,381.9,379.7],
                                    [382.7,379.2,381.7,379.8],
                                    [382.7,379.1,381.7,379.9],
                                    [382.7,379.1,381.7,379.9],
                                    [382.7,379.1,382,380],
                                    [382.8,379,382.1,379.9],
                                    [382.8,379,381.8,380.1],
                                    [382.8,379.1,381.7,380.1],
                                    [382.7,378.9,381.9,380.1],
                                    [382.9,378.8,382,380.3],
                                    [382.9,378.8,381.9,380.3],
                                    [383.7,378.6,381.8,380.5],
                                    [383.2,378.4,381.7,380.6],
                                    [382.8,378.4,381.8,380.7],
                                    [383,378.4,381.7,380.7],
                                    [383.1,378.2,381.8,380.9],
                                    [383.2,378.1,382,380.8],
                                    [383.1,378.2,381.9,380.7],
                                    [383,378.2,381.7,380.7],
                                    [382.9,378.3,381.9,380.6],
                                    [383,378.5,381.9,380.5],
                                    [382.9,378.6,382.1,380.4],
                                    [382.8,378.7,382.1,380.3],
                                    [382.8,378.8,382,380.3],
                                    [382.7,378.7,382,380.2],
                                    [382.9,378.7,381.9,380.4],
                                    [383,378.5,381.7,380.4],
                                    [383,378.4,382.2,380.6],
                                    [383,378.4,381.9,380.6],
                                    [383.2,378.2,381.8,380.8],
                                    [383.1,378.3,381.7,380.9],
                                    [383.1,378.1,381.7,380.8],
                                    [383.3,378.1,381.5,380.9],
                                    [383.2,378.1,382,380.8],
                                    [383.3,378.1,381.9,381],
                                    [383.3,378,381.7,381],
                                    [383.4,377.9,381.4,380.9],
                                    [383.3,377.9,381.4,381],
                                    [383.4,378,381.6,381],
                                    [383.3,378,381.7,381],
                                    [383.4,378,381.9,381],
                                    [383.3,378,381.5,381],
                                    [383.3,377.9,381.6,381],
                                    [383.3,377.8,382,381.1],
                                    [383.3,377.9,382,381],
                                    [383.4,377.7,381.9,381.3],
                                    [383.4,377.7,381.9,381.3],
                                    [383.4,377.7,382.1,381.3],
                                    [383.3,377.6,382,381.3],
                                    [383.4,377.8,381.9,381.3],
                                    [383.3,377.6,381.7,381.4],
                                    [383.3,377.7,382,381.4],
                                    [383.3,377.7,382.1,381.3],
                                    [383.3,377.7,382.1,381.3],
                                    [383.2,377.8,381.8,381.2],
                                    [383.2,378,382.1,381.1],
                                    [383.1,378.3,382.1,380.9],
                                    [383,378.4,382.1,380.7],
                                    [383.1,378.2,382,380.8],
                                    [383,378.1,382.1,381],
                                    [383,378,382.3,381.1],
                                    [383,378,382,381.2],
                                    [383,377.9,382.1,381.3],
                                    [383,378,382,381.4],
                                    [383,377.8,382.2,381.4],
                                    [383,377.8,382.5,381.5],
                                    [383,377.8,382.4,381.6],
                                    [383.1,377.8,382.3,381.5],
                                    [383.2,377.8,382.4,381.6],
                                    [383.1,377.8,381.9,381.8],
                                    [383,377.7,382,381.9],
                                    [383,377.7,382.2,381.9],
                                    [383.1,377.8,382.2,382],
                                    [383.1,377.7,382.3,382.2],
                                    [383.1,377.7,382.2,382.3],
                                    [383.2,377.6,382.1,382.4],
                                    [383.2,377.6,382.2,382.5],
                                    [383.2,377.6,382.4,382.7],
                                    [383.3,377.7,382.4,382.8],
                                    [383.3,377.7,382.2,382.9],
                                    [383.4,377.5,382.1,383.1],
                                    [383.4,377.5,382.2,383.3],
                                    [383.5,377.6,382.1,383.6],
                                    [383.4,377.5,382.3,383.7],
                                    [383.6,377.3,382.2,383.8],
                                    [383.6,377.2,382.2,384],
                                    [383.6,377.3,382.2,384],
                                    [383.6,377.2,382.3,384.2],
                                    [383.7,377.2,382.3,384.5],
                                    [383.8,377.1,382.3,384.6],
                                    [383.8,377,382.3,384.8],
                                    [383.9,376.9,382.2,384.8],
                                    [384,376.8,382.2,384.9],
                                    [384,376.8,381.8,385.1],
                                    [384.1,376.8,381.9,385.2],
                                    [384.1,376.7,382,385.3],
                                    [384.2,376.6,381.8,385.4],
                                    [384.2,376.6,381.9,385.5],
                                    [384.4,376.6,381.8,385.6],
                                    [384.4,376.6,381.9,385.7],
                                    [384.5,376.4,381.6,385.8],
                                    [384.5,376.4,381.7,385.9],
                                    [384.3,376.3,381.8,386],
                                    [384.1,376.2,381.8,386.1],
                                    [384.1,376.3,381.7,386.1],
                                    [384.2,376.1,381.8,386.4],
                                    [384.2,376.1,381.9,386.5],
                                    [384.3,375.9,381.7,386.4],
                                    [384.4,375.8,381.8,386.6],
                                    [384.6,376,381.6,386.6],
                                    [384.5,375.9,381.6,386.7],
                                    [384.5,375.8,381.5,386.9],
                                    [384.5,375.5,381.5,386.9],
                                    [384.6,375.6,381.5,386.9],
                                    [384.7,375.6,381.4,387],
                                    [384.6,375.6,381.7,386.9],
                                    [384.8,375.6,381.6,387.1],
                                    [384.6,375.4,381.3,387.2],
                                    [384.7,375.3,381.5,387.1],
                                    [384.5,375.3,381.5,387.1],
                                    [384.5,375.3,381.6,387.2],
                                    [384.5,375.2,381.5,387.2],
                                    [384.5,375.3,381.4,387.2],
                                    [384.6,375.3,381.2,387.3],
                                    [384.6,375.3,381.3,387.2],
                                    [384.5,375.2,381.4,387.3],
                                    [384.5,375.3,381.5,387.3],
                                    [384.5,375.2,381.2,387.3],
                                    [384.6,375.1,381.2,387.4],
                                    [384.5,375.3,381.3,387.4],
                                    [384.5,375.2,381.2,387.4],
                                    [384.5,375.2,381.2,387.3],
                                    [384.4,375.3,381.3,387.3],
                                    [384.4,375.3,381.2,387.4],
                                    [384.5,375.2,381.5,387.5],
                                    [384.5,375.2,381.2,387.3],
                                    [384.4,375.2,381.3,387.3],
                                    [384.5,375.1,381.4,387.3],
                                    [384.5,375.1,381.3,387.4],
                                    [384.4,375.1,381.3,387.3],
                                    [384.5,375,381.2,387.3],
                                    [384.4,374.9,380.9,387.3],
                                    [384.5,374.9,381,387.3],
                                    [384.5,374.9,381.1,387.4],
                                    [384.5,374.8,381.3,387.3],
                                    [384.4,374.7,381.4,387.3],
                                    [384.4,374.8,381.3,387.4],
                                    [384.4,374.8,381.4,387.5],
                                    [384.3,374.7,381.4,387.4],
                                    [384.3,374.6,381.1,387.5],
                                    [384.3,375.2,381.2,386.9],
                                    [384.2,374.7,381.3,387.3],
                                    [384.4,374.9,381.1,387.2],
                                    [384,374.6,381.7,387.3],
                                    [384.3,374.4,381.4,387.6],
                                    [384.2,375.3,381.4,386.6],
                                    [383.7,374.8,381.9,387],
                                    [383.8,374.8,381.9,387],
                                    [383.8,374.7,381.9,387.1],
                                    [383.8,374.4,381.8,387.3],
                                    [383.7,374.4,381.6,387.2],
                                    [383.8,374.2,381.6,387.4],
                                    [383.8,374.2,381.5,387.4],
                                    [383.8,374.1,381.6,387.4],
                                    [383.9,374,381.8,387.4],
                                    [383.8,374.1,381.8,387.3],
                                    [383.8,374.1,381.7,387.4],
                                    [383.8,374.1,381.7,387.4],
                                    [383.8,373.9,381.6,387.4],
                                    [383.8,373.7,381.9,387.6],
                                    [383.8,374,381.8,387.4],
                                    [384.2,372.8,381.6,388.4],
                                    [384,373,381.6,388.1],
                                    [384.2,372.8,381.5,388.4],
                                    [383.9,373.1,381.8,388.1],
                                    [384,373,381.7,388.1],
                                    [384,372.8,381.6,388.2],
                                    [384,372.7,381.6,388.2],
                                    [384.2,372.3,381.6,388.6],
                                    [384.3,372.4,381.5,388.4],
                                    [384.5,371.6,381.5,389.1],
                                    [384.4,371.7,381.6,389.1],
                                    [384.5,371.3,381.4,389.4],
                                    [384.5,371.4,381.4,389.2],
                                    [384.6,371.3,381.3,389.4],
                                    [384.6,371.3,381.5,389.5],
                                    [384.7,371.1,381.2,389.5],
                                    [384.8,370.9,381.3,389.7],
                                    [384.6,371,381.3,389.6],
                                    [384.5,371,381.4,389.5],
                                    [384.6,370.8,381.4,389.7],
                                    [384.9,370.5,381.2,390.1],
                                    [384.5,370.6,381.5,389.9],
                                    [384.8,370.3,381.2,390.4],
                                    [384.8,370,381.3,390.5],
                                    [384.8,370.2,381.4,390.4],
                                    [384.9,369.9,381.4,390.8],
                                    [384.7,370.2,381.4,390.1],
                                    [384.8,370.1,381.4,390.3],
                                    [384.6,370.6,381.4,389.8],
                                    [384.5,370.8,381.4,389.6],
                                    [384.5,370.8,381.4,389.6],
                                    [384.7,370.5,381.3,389.8],
                                    [384.5,370.7,381.3,389.7],
                                    [384.6,370.7,381.3,389.6],
                                    [384.6,370.4,381.3,389.7],
                                    [384.9,369.9,381.2,390.4],
                                    [384.9,370.3,381.2,390.1],
                                    [384.4,371.1,381.5,389.4],
                                    [384.7,371,381.1,389.4],
                                    [384.5,371,381.1,389.3],
                                    [384.4,371.5,381.1,388.9],
                                    [384.8,370.8,381.1,389.7],
                                    [384.6,370.9,381.2,389.4],
                                    [384.7,371,381,389.3],
                                    [384.8,370.6,381,389.7],
                                    [384.8,370.9,381,389.7],
                                    [384.7,371.1,381,389.4],
                                    [384.7,370.8,381.1,389.7],
                                    [384.7,371,380.8,389.5],
                                    [384.6,371.3,381,389.2],
                                    [384.8,370.8,381,389.8],
                                    [384.9,371.2,380.7,389.5],
                                    [384.8,371.4,380.9,389.2],
                                    [384.3,371,381.2,389.4],
                                    [384.5,370.5,381.1,389.9],
                                    [385.4,371.2,380.2,389.7],
                                    [384.7,371.5,380.9,389.1],
                                    [384.7,370.4,380.9,389.8],
                                    [385.4,371.1,380.2,389.6],
                                    [384.9,371.3,380.7,389.2],
                                    [384.6,370.3,380.9,389.9],
                                    [384.9,369.8,380.9,390.3],
                                    [385.6,370.4,380,389.9],
                                    [385,370.6,380.4,389.5],
                                    [385.1,369.9,380.8,390.2],
                                    [385.5,370.7,380.1,389.7],
                                    [385.2,370.7,380.3,389.5],
                                    [385,370.2,380.6,389.9],
                                    [385.4,370.7,380.1,389.7],
                                    [385.1,370.7,380.4,389.6],
                                    [385.1,370.2,380.6,390.1],
                                    [385.5,370.4,380.2,390.1],
                                    [385.2,370.9,380.4,389.5],
                                    [385,370.1,380.9,390.1],
                                    [385.1,369.9,380.7,390.3],
                                    [385.4,370.8,380,389.8],
                                    [384.9,371.3,380.3,389],
                                    [384.9,370.7,380.6,389.6],
                                    [385.3,370.6,380.2,389.8],
                                    [385.2,371.1,380.2,389.5],
                                    [384.8,371.8,380.5,388.7],
                                    [384.6,371.2,380.6,389.2],
                                    [384.5,370.9,380.9,389.3],
                                    [384.6,370.4,380.7,389.7],
                                    [385.3,371.4,379.8,389.2],
                                    [384.8,372,380.3,388.3],
                                    [384.5,371.7,380.6,388.6],
                                    [384.3,371.6,380.8,388.7],
                                    [384.3,371.1,380.9,389.1],
                                    [384.3,371.1,380.8,389.1],
                                    [384.6,371.1,380.5,389.3],
                                    [384.8,371.1,380.5,389.2],
                                    [384.9,371,380.6,389.3],
                                    [384.9,371.1,380.2,389.3],
                                    [385,371.2,380.2,389.2],
                                    [384.9,371.3,380.2,389.1],
                                    [385,371.4,380.2,389.1],
                                    [384.9,371.5,380.2,388.9],
                                    [384.9,371.7,380.2,388.7],
                                    [385,371.8,380,388.6],
                                    [385,371.7,380.1,388.6],
                                    [384.8,372.1,380,388.2],
                                    [384.7,372.2,380.2,388.2],
                                    [384.8,372.1,380.2,388.3],
                                    [385,372,379.9,388.4],
                                    [385,372,379.9,388.5],
                                    [385.1,371.8,379.9,388.6],
                                    [385.2,371.7,379.8,388.8],
                                    [385.2,371.7,379.9,388.6],
                                    [385.3,371.7,379.9,388.6],
                                    [385.4,371.6,379.8,388.7],
                                    [385.5,371.8,379.8,388.7],
                                    [385.4,371.8,379.8,388.8],
                                    [385.5,371.6,379.2,388.7],
                                    [385.5,371.6,379.5,388.7],
                                    [385.4,371.8,379.6,388.6],
                                    [385.6,371.6,379.4,388.8],
                                    [385.6,371.7,379.3,388.7],
                                    [385.7,371.9,379.1,388.6],
                                    [385.8,372.1,379.3,388.5],
                                    [385.9,372.1,379.3,388.5],
                                    [386,372.1,379,388.4],
                                    [385.9,372.2,379,388.4],
                                    [386,372,378.9,388.5],
                                    [385.9,371.8,379.1,388.6],
                                    [386,371.9,379.2,388.6],
                                    [385.9,371.8,379,388.6],
                                    [385.9,371.8,379,388.7],
                                    [385.9,371.9,379.3,388.7],
                                    [386,371.9,378.9,388.7],
                                    [386.1,371.7,378.9,388.7],
                                    [386,371.8,378.9,388.6],
                                    [386.1,371.9,378.9,388.6],
                                    [386.1,371.9,378.8,388.6],
                                    [386.2,371.8,378.9,388.6],
                                    [386.1,371.9,378.9,388.6],
                                    [386.2,371.8,378.8,388.6],
                                    [386.2,371.9,378.9,388.6],
                                    [386.3,371.9,378.6,388.6],
                                    [386.3,371.9,378.7,388.7],
                                    [386.4,372,378.7,388.6],
                                    [386.4,371.9,378.6,388.6],
                                    [386.5,372,378.5,388.6],
                                    [386.5,372,378.4,388.6],
                                    [386.5,372,378.2,388.5],
                                    [386.7,372,378.3,388.5],
                                    [386.7,372,378.2,388.5],
                                    [386.7,372,378.1,388.5],
                                    [386.9,372,377.9,388.6],
                                    [387,372.1,378.1,388.6],
                                    [387.1,372,377.9,388.8],
                                    [387,372,377.8,388.6],
                                    [387.2,372,377.9,388.7],
                                    [387.1,372.1,377.7,388.6],
                                    [387.2,372.1,377.8,388.7],
                                    [387.2,372.1,377.5,388.6],
                                    [387.2,372.2,377.5,388.6],
                                    [387.4,372.1,377.3,388.7],
                                    [387.5,372.1,377.3,388.7],
                                    [387.5,372.1,377.7,388.7],
                                    [387.5,372,377.2,388.7],
                                    [387.6,372,377.4,388.8],
                                    [387.6,372,377.4,388.7],
                                    [387.6,372.1,377.4,388.8],
                                    [387.7,372,377.3,388.8],
                                    [387.8,371.9,377.3,388.8],
                                    [387.7,371.9,377.2,388.9],
                                    [387.6,372,377.2,388.8],
                                    [387.7,371.8,377.2,388.9],
                                    [387.7,371.8,377,388.9],
                                    [193.5,198.5,192.5,190.1]];
    !
!   CONST robtarget pOrigin:=[[0,0,0],[1,0,0,0],[0,0,1,1],[8200,9E+09,9E+09,9E+09,9E+09,9E+09]];
 !   PERS robtarget pOrigin:=[[0,0,0],[1,0,0,0],[0,-1,0,0],[2253.54,9E+09,9E+09,9E+09,9E+09,9E+09]];
!    CONST robtarget pOrigin:=[[0,0,0],[1,0,0,0],[-1,0,1,0],[5500,9E+09,9E+09,9E+09,9E+09,9E+09]];
!    CONST robtarget pOrigin:=[[0,0,0],[1,0,0,0],[-1,0,2,0],[6500,9E+09,9E+09,9E+09,9E+09,9E+09]];

!    PERS robtarget pOrigin:=[[0,0,0],[1,0,0,0],[0,-2,1,0],[0,9E+9,9E+9,9E+9,9E+9,9E+9]];
    CONST zonedata zone01:=[FALSE,0.001,0.001,0.1,0.01,0.1,0.1];
    !
    PERS pos posCenterTube:=[-15.6158,675.69,271.899];
    PERS pos posDelta:=[-3,0,4.14999];
!    PERS robtarget pActualCalc:=[[-991.421,1033.05,-83.7236],[0.999887,-0.00648616,8.80107E-05,-0.0135675],[0,-1,1,0],[0,9E+09,9E+09,9E+09,9E+09,9E+09]];
    PERS pos pnewCalc:=[-0.770965,0,57.4255];

    PROC rPathFollowSystemPreStart()
        !
        END_TUBE_REACHED:=[FALSE, FALSE];
        nMovementCounter:=1;
        rCalcCenterPointTube;
        !
        TargetNew{CALC_COUNTER+nMovementCounter}:=TargetNew{1};
        TargetNew{CALC_COUNTER+nMovementCounter}.trans:=posCenterTube;
        !
!        Maak tussen de eerste berekende CP en startpunt een lineaire lijn voor beweegrichting
        reg1:=(TargetNew{CALC_COUNTER+nMovementCounter}.trans.x-TargetNew{nMovementCounter}.trans.x)/CALC_COUNTER;
        reg2:=(TargetNew{CALC_COUNTER+nMovementCounter}.trans.y-TargetNew{nMovementCounter}.trans.y)/CALC_COUNTER;
        reg3:=(TargetNew{CALC_COUNTER+nMovementCounter}.trans.z-TargetNew{nMovementCounter}.trans.z)/CALC_COUNTER;
!        Vul deze positie in de eerste reeks datapunten in
        FOR i FROM 2 TO CALC_COUNTER DO
            TargetNew{i}:=TargetNew{i-1};
            TargetNew{i}.trans.x:=TargetNew{i}.trans.x+reg1;
            TargetNew{i}.trans.y:=TargetNew{i}.trans.y+reg2;
            TargetNew{i}.trans.z:=TargetNew{i}.trans.z+reg3;
        ENDFOR
        !
        WHILE nMovementCounter<PreStartLength DO
!            Start movement
            Incr nMovementCounter;
            MoveL Reltool(TargetNew{nMovementCounter},0,0,0),v20,Zone01,tInductionRing\WObj:=wTempClamp;
                        !
            rCalcCenterPointTube;
            !
            TargetNew{CALC_COUNTER+nMovementCounter}:=TargetNew{1};
            TargetNew{CALC_COUNTER+nMovementCounter}.trans:=posCenterTube;
            !
            rLinearFilter;
        ENDWHILE
        ! bereken op basis van deze 100 datapunten een nieuw startpositie
        rCalcStartPos;
        !
        ! op bais van deze rechte lijn hoort een orientatie, dit is de start orientatie
        rCalcOrient;
        !
        TargetNew{1}.rot:=TargetNew{nOrientFilterCounter}.rot;
        !
        ! beweeg retour naar nieuw bepaalde start positie

        MoveL Reltool(TargetNew{1},0,0,0), v20, Zone01, tInductionRing\WObj:=wTempClamp;
        !
        ! de berekende orientatie overnemen voor de eerste 100 datapunten
        FOR i FROM 1 TO 95 DO
            TargetNew{i}.rot:=TargetNew{1}.rot;
        ENDFOR
        !
    ENDPROC

    PROC rPathFollowSystem()
        !
        nLaserOutRange{1} := 0;
        nLaserOutRange{2} := 0;
        nLaserOutRange{3} := 0;
        nLaserOutRange{4} := 0;
        !
!        nMovementCounter:=1;
        rCalcCenterPointTube;
        !
        TargetNew{CALC_COUNTER+nMovementCounter}:=TargetNew{1};
        TargetNew{CALC_COUNTER+nMovementCounter}.trans:=posCenterTube;
        !
        WHILE (nMovementCounter<4000 AND END_TUBE_REACHED{1}=FALSE AND END_TUBE_REACHED{2}=FALSE) AND diRequestStopReceived=0 DO
            Incr nMovementCounter;


!            IF OFFSET<>offsetprev THEN
!                MoveL Reltool(TargetNew{nMovementCounter-1},OFFSET.x,0,OFFSET.z\Ry:=-10),v5000,Zone01,tInductionRing\WObj:=wTempClamp;
!            ENDIF
            !
            offsetprev:=OFFSET;
            rTrackPosition;

            !OFFSET := bound(OFFSET_REF, OFFSET + sign(OFFSET_REF-OFFSET)*vmax*dt);
!            reg1 := ((OFFSET_REF.x-OFFSET.x)/abs(OFFSET_REF.x-OFFSET.x));
!            reg2 := max(abs(OFFSET_REF.x-OFFSET_REF), reg1*10)
!            IF reg1>0       OFFSET.x := max(OFFSET_REF.x, OFFSET.x + reg1*10);
!            IF reg1<0       OFFSET.x := max(OFFSET_REF.x, OFFSET.x + reg1*10);




            MoveL Reltool(TargetNew{nMovementCounter},OFFSET.x,0,OFFSET.z),v10,Zone01,tInductionRing\WObj:=wTempClamp;
            !
            rCalcCenterPointTube;
            !
            TargetNew{CALC_COUNTER+nMovementCounter}:=TargetNew{1};
            TargetNew{CALC_COUNTER+nMovementCounter}.trans:=posCenterTube;
            TargetNew{CALC_COUNTER+nMovementCounter}.robconf:=pConfigCopy.robconf;
            !
            rLinearFilter;
            !
            rCalcOrient;
            !
            rTubeEnd;
        ENDWHILE
        !
        Waittime 1;
        TPErase;
        IF END_TUBE_REACHED{1} THEN
            TPWrite "END_TUBE_REACHED TUBE DIAMETER CHANGE";
        ENDIF
        IF END_TUBE_REACHED{2} THEN
            TPWrite "END_TUBE_REACHED SENSOR OUT RANGE";
        ENDIF
        TPWrite "END_TUBE_REACHED";
        TPWrite "MovementCounter =  "\num:=nMovementCounter;
        nLastIdentifiedTarget:=nMovementCounter;

        !
        Waittime 5;
        !
    ENDPROC

    PROC rFreeRunFwd()
        WHILE nMovementCounter<nLastIdentifiedTarget DO
            Incr nMovementCounter;
            MoveL Reltool(TargetNew{nMovementCounter},OFFSET.x,0,OFFSET.z),v20,Zone01,tInductionRing\WObj:=wTempClamp;
        ENDWHILE
        !
        !TPWrite "ENDT_TUBE_REACHED";
        !TPWrite "MovementCounter =  "\num:=nMovementCounter;
        !Stop;
    ENDPROC

    PROC rFreeRunBwd(bool HeatTreatment)
        VAR speeddata Speeddummy;

        IF HeatTreatment THEN

        ENDIF
        Speeddummy:=v50;
        WHILE nMovementCounter>=2 DO
            Decr nMovementCounter;
            IF nMovementCounter<5       Speeddummy:=v50;
            MoveL Reltool(TargetNew{nMovementCounter},OFFSET.x,0,OFFSET.z), Speeddummy, Zone01, tInductionRing\WObj:=wTempClamp;
        ENDWHILE
        !
        TPWrite "START_TUBE_REACHED";
        TPWrite "MovementCounter =  "\num:=nMovementCounter;
        !Stop;
    ENDPROC
ENDMODULE
